Staubli VAL3: childAction.pgx

public program childAction(viewType& view, num& rootItem_, num& childItem_, num keyCode_)
begin
end
